(* CoDeSys 2.3.9.42 project: Preobrazovatel_83.pro *)

(* POU PLC_PRG, ST *)
PROGRAM PLC_PRG
VAR
	tok_low:REAL:=4;
	tok_high:REAL:=20;
	diap_low,diap_high :REAL; (*диапазоны измеряемой температуры *)
	Tok : REAL ; (*ток 4-20 мА*)
	Prom : REAL ; (*промежеточная переменная*)
	Lamp1: BOOL; (*лампа, выход за диапазон градусов*)
	Temp1 : REAL ; (*температура*)
END_VAR
Lamp1 := (Tok > tok_high) OR (Tok < tok_low) ;

Prom:=LIMIT(tok_low, Tok, tok_high);

Temp1:=((diap_high*(Prom-4))/16);
END_PROGRAM
